// TIA Portal V16 export
// export: Created 2022-02-11T09:26:12.5858984Z, ExportSetting WithDefaults, DisplayName Totally Integrated Automation Portal, DisplayVersion V16 Update 5, DisplayName TIA Portal Version Control Interface, DisplayVersion V16 Update 2, DisplayName TIA Portal Openness, DisplayVersion V16 Update 5, DisplayName STEP 7 Professional, DisplayVersion V16 Update 5, DisplayName STEP 7 Safety, DisplayVersion V16, DisplayName WinCC Professional, DisplayVersion V16 Update 5, DisplayName SIMATIC Visualization Architect, DisplayVersion V16
VAR_GLOBAL   // PLC tag table "Tabla de variables estándar"
END_VAR
